// Binary Controller
FUNCTION_BLOCK FB_CRYO_BIN_CTRL
VAR_INPUT
	in_nFeedback:		E_CRYO_BIN_ACT_FEEDBACK := E_CRYO_BIN_ACT_FEEDBACK.ON_ONLY;	// Feedbacks
	in_nTimeout:		UDINT := 10000;	// Timeout for switching on/off [ms]. Default 10000.
	in_bActiveLowCtrl:	BOOL := FALSE;	// Active Low for Control output
	in_bActiveLowStat:	BOOL := FALSE;	// Active Low for Status signals, i.e. feedback
	in_bEnable:			BOOL := FALSE;	// Controller active while in_bEnable is TRUE
END_VAR
VAR
	
	{attribute 'OPC.UA.DA' := '1'}
	Actuator:	FB_CRYO_BIN_ACT;	// Heater, valve, etc.
	
	stat:		T_CRYO_BIN_CTRL_STATUS;


	{attribute 'OPC.UA.DA' := '0'}
	bReset:		BOOL := FALSE;		// RESET Command


	{attribute 'OPC.UA.DA' := '0'}
	timer:		TON;		// Timer for commands
	
	
END_VAR

// Increment cycle counter
stat.nCycleCounter := stat.nCycleCounter + 1;

// Execute Actuator FB on every cycle
Actuator(
	in_nFeedback		:= in_nFeedback,
	in_nTimeout			:= in_nTimeout,
	in_bActiveLowCtrl	:= in_bActiveLowCtrl,
	in_bActiveLowStat	:= in_bActiveLowStat);


CASE stat.nState OF
	/////////////////////////////////
	E_CRYO_BIN_CTRL_STATE.NONE:
	/////////////////////////////////
	//
	// This is the state on power-up.
	// Determine the initial state based on the command amd actuator state.
	IF Actuator.stat.bError  OR NOT stat.bCtrlOK	THEN
		stat.nState	:= E_CRYO_BIN_CTRL_STATE.ERROR;
	ELSIF in_bEnable  AND  Actuator.stat.bON	THEN
		stat.nState	:= E_CRYO_BIN_CTRL_STATE.ACTIVE_ON;
	ELSIF in_bEnable  AND  Actuator.stat.bOFF	THEN
		stat.nState	:= E_CRYO_BIN_CTRL_STATE.ACTIVE_OFF;
	ELSIF NOT in_bEnable  THEN
		stat.nState	:= E_CRYO_BIN_CTRL_STATE.OFF;
	END_IF
	M_SetStatus(stat.nState);	
	RETURN;
	

	/////////////////////////////////
	E_CRYO_BIN_CTRL_STATE.OFF:
	/////////////////////////////////
	//
	IF	Actuator.stat.bError	OR NOT stat.bCtrlOK	THEN
		stat.nState	:= E_CRYO_BIN_CTRL_STATE.ERROR;
	ELSIF in_bEnable  THEN
		// Activate the control loop.
		// Goto Active_Off first.
		//
		// Start the timer
		timer(IN:=FALSE);
		timer(IN:=TRUE, PT:=UDINT_TO_TIME(in_nTimeout));
		// Set next state
		stat.nState	:= E_CRYO_BIN_CTRL_STATE.ACTIVE_OFF;
	END_IF
	M_SetStatus(stat.nState);	
	RETURN;
	
	
	/////////////////////////////////
	E_CRYO_BIN_CTRL_STATE.ACTIVE_OFF:
	/////////////////////////////////
	//
	IF	Actuator.stat.bError	OR NOT stat.bCtrlOK  THEN
		stat.nState	:= E_CRYO_BIN_CTRL_STATE.ERROR;
	ELSIF NOT in_bEnable  THEN
		// Goto Off.
		//
		// Set next state
		stat.nState	:= E_CRYO_BIN_CTRL_STATE.OFF;
	ELSIF M_User_SetAction() = E_CRYO_BIN_CTRL_ACTION.ON THEN
		// Goto Active_Off.
		//
		// Start the timer
		timer(IN:=FALSE);
		timer(IN:=TRUE, PT:=UDINT_TO_TIME(in_nTimeout));
		
		// Trigger action
		Actuator(in_bExecute:=FALSE);
		Actuator(in_bExecute:=TRUE, in_nCommand:=E_CRYO_BIN_ACT_CMD.ON);
		
		// Set next state
		stat.nState	:= E_CRYO_BIN_CTRL_STATE.ACTIVE_SWITCHING_ON;
	END_IF
	M_SetStatus(stat.nState);	
	RETURN;
	
	
	//////////////////////////////////////////
	E_CRYO_BIN_CTRL_STATE.ACTIVE_SWITCHING_ON:
	//////////////////////////////////////////
	//
	// Check for timeout
	timer(IN:=TRUE);
	IF timer.Q THEN
		// Stop the timer
		timer(IN:=FALSE);
		// Goto ERROR state
		stat.nState	:= E_CRYO_BIN_CTRL_STATE.ERROR;
	ELSIF	Actuator.stat.bError	THEN
		stat.nState	:= E_CRYO_BIN_CTRL_STATE.ERROR;
	ELSIF Actuator.stat.bON THEN
		// The actuator is ON, transition completed.
		// Goto Active_On.
		stat.nState	:= E_CRYO_BIN_CTRL_STATE.ACTIVE_ON;
	END_IF
	M_SetStatus(stat.nState);	
	RETURN;
	

	/////////////////////////////////
	E_CRYO_BIN_CTRL_STATE.ACTIVE_ON:
	/////////////////////////////////
	//
	IF	Actuator.stat.bError	THEN
		stat.nState	:= E_CRYO_BIN_CTRL_STATE.ERROR;
	ELSIF	NOT in_bEnable 		OR  
			NOT stat.bCtrlOK	OR
			M_User_SetAction() = E_CRYO_BIN_CTRL_ACTION.OFF THEN
		// Goto Active_Off.
		// If NOT in_bExecute, the system will continue to complete OFF
		//
		// Start the timer
		timer(IN:=FALSE);
		timer(IN:=TRUE, PT:=UDINT_TO_TIME(in_nTimeout));
		
		// Trigger action
		Actuator(in_bExecute:=FALSE);
		Actuator(in_bExecute:=TRUE, in_nCommand:=E_CRYO_BIN_ACT_CMD.OFF);
		
		// Set next state
		stat.nState	:= E_CRYO_BIN_CTRL_STATE.ACTIVE_SWITCHING_OFF;
	END_IF
	M_SetStatus(stat.nState);	
	RETURN;
	
	
	///////////////////////////////////////////
	E_CRYO_BIN_CTRL_STATE.ACTIVE_SWITCHING_OFF:
	///////////////////////////////////////////
	//
	// Check for timeout
	timer(IN:=TRUE);
	IF timer.Q THEN
		// Stop the timer
		timer(IN:=FALSE);
		// Goto ERROR state
		stat.nState	:= E_CRYO_BIN_CTRL_STATE.ERROR;
	ELSIF	Actuator.stat.bError	THEN
		stat.nState	:= E_CRYO_BIN_CTRL_STATE.ERROR;
	ELSIF Actuator.stat.bOFF THEN
		// The actuator is OFF, transition completed.
		// Goto Active_Off.
		stat.nState	:= E_CRYO_BIN_CTRL_STATE.ACTIVE_OFF;
	END_IF
	M_SetStatus(stat.nState);	
	RETURN;
	
	/////////////////////////////////
	E_CRYO_BIN_CTRL_STATE.ERROR:
	/////////////////////////////////
	//
	M_User_TryRecovery();

END_CASE

METHOD M_Reset
VAR_INPUT
END_VAR
// By setting the bReset flag,
// The actuator will try to exit error state.
// In ERROR state, method M_User_TryRecovery() is executed.
bReset	:= TRUE;
END_METHOD

METHOD M_SetStatus
VAR_INPUT
	nState:	E_CRYO_BIN_CTRL_STATE;
END_VAR
stat.bActON		:= Actuator.stat.bON;
stat.bActOFF	:= Actuator.stat.bOFF;


CASE nState OF
	
	E_CRYO_BIN_CTRL_STATE.OFF:
	stat.bDone	:= TRUE;
	stat.bBusy	:= FALSE;
	stat.bError	:= FALSE;
	stat.bActive:= FALSE;
	stat.sState	:= 'OFF';
	
	E_CRYO_BIN_CTRL_STATE.ACTIVE_OFF:
	stat.bDone	:= TRUE;
	stat.bBusy	:= FALSE;
	stat.bError	:= FALSE;
	stat.bActive:= TRUE;
	stat.sState	:= 'ACTIVE_OFF';
	
	E_CRYO_BIN_CTRL_STATE.ACTIVE_ON:
	stat.bDone	:= TRUE;
	stat.bBusy	:= FALSE;
	stat.bError	:= FALSE;
	stat.bActive:= TRUE;
	stat.sState	:= 'ACTIVE_ON';
	
	E_CRYO_BIN_CTRL_STATE.ACTIVE_SWITCHING_ON:
	stat.bDone	:= FALSE;
	stat.bBusy	:= TRUE;
	stat.bError	:= FALSE;
	stat.bActive:= TRUE;
	stat.sState	:= 'ACTIVE_SWITCHING_ON...';
	
	E_CRYO_BIN_CTRL_STATE.ACTIVE_SWITCHING_OFF:
	stat.bDone	:= FALSE;
	stat.bBusy	:= TRUE;
	stat.bError	:= FALSE;
	stat.bActive:= TRUE;
	stat.sState	:= 'ACTIVE_SWITCHING_OFF...';
	
	E_CRYO_BIN_CTRL_STATE.ERROR:
	stat.bDone	:= TRUE;
	stat.bBusy	:= FALSE;
	stat.bError	:= TRUE;
	stat.bActive:= FALSE;
	stat.sState	:= 'ERROR';

END_CASE
END_METHOD

METHOD M_User_SetAction : INT
VAR_INPUT
END_VAR
// TODO USER
//
// This method implements the logic for controlling the actuator.
// The actuator can be a heater, valve, etc.
// There are two input values from sensors and two deltas for comparison.
//
// This example implements the heater control with the following assumptions:
//
// in_lrInput1 - Temperature of the Cryo Bench (B)
// in_lrInput2 - Temperature of the Detector (D). Coming from Lakeshore.
// in_lrPar1 - Delta [K] to turn the heater ON:  IF B < D - in_lrPar1
// in_lrPar2 - Delta [K] to turn the heater OFF: IF B > D - in_lrPar2
//
// in_lrDelta1 > in_lrDelta2, e.g. 10K > 4K.
//
IF	stat.nState = E_CRYO_BIN_CTRL_STATE.ACTIVE_OFF  OR  
	stat.nState = E_CRYO_BIN_CTRL_STATE.ACTIVE_ON THEN
(*	
	IF in_lrInput1 < in_lrInput2 - in_lrPar1 THEN
		// Activate the actuator
		M_User_SetOutput	:= E_CRYO_BIN_CTRL_ACTION.ON;
	ELSIF in_lrInput1 > in_lrInput2 - in_lrPar2 THEN
		// Dectivate the actuator
		M_User_SetOutput	:= E_CRYO_BIN_CTRL_ACTION.OFF;
	END_IF
*)
ELSE
	// Don't do anything
	M_User_SetAction	:= E_CRYO_BIN_CTRL_ACTION.NONE;
END_IF
END_METHOD

METHOD M_User_TryRecovery
VAR_INPUT
END_VAR
// TODO USER
// This is the default recovery routine.
// To be customided by the user, if needed.
//
IF bReset THEN
	// RESET the controller in order to try to clear error
	bReset	:= FALSE;	// Clear RESET flag
	
	// Start the timer
	timer(IN:=FALSE);
	timer(IN:=TRUE, PT:=T#5S);
	
	// Trigger action
	Actuator(in_bExecute:=FALSE);
	Actuator(in_bExecute:=TRUE, in_nCommand:=E_CRYO_BIN_ACT_CMD.OFF);
	
	// Goto SWITCHING_OFF state
	stat.nState	:= E_CRYO_BIN_CTRL_STATE.ACTIVE_SWITCHING_OFF;
	M_SetStatus(stat.nState);	
ELSIF NOT Actuator.stat.bError AND stat.bCtrlOK  THEN
	// Self recovery since everything seems to be OK now.
	// Goto NONE state.
	// From there proper state will be found and set.
	stat.nState	:= E_CRYO_BIN_CTRL_STATE.NONE;
	M_SetStatus(stat.nState);	
END_IF
END_METHOD

END_FUNCTION_BLOCK

(* stored: Version 1.1.0.1, ProductVersion 3.1.4024.12
   POU FB_CRYO_BIN_CTRL: Id {911ba4c8-b9f4-47c8-a937-6e4327965c35}, SpecialFunc None
   Method M_Reset: Id {5e9e5b69-a092-4050-96d5-b4c0bb6fb059}
   Method M_SetStatus: Id {89312a00-5c08-4e45-9d98-831d0a6b2667}
   Method M_User_SetAction: Id {ec97d002-202c-4612-975b-6d9857b07066}
   Method M_User_TryRecovery: Id {b466d6fe-28bb-4b23-a093-43ae31684784} *)
